TYPE U_NCI_R_PARAMETER_I :
UNION

  stCtrl              : ARRAY[1..MAX_NCI_CH] OF ST_R_Parameter;

  byCtrl    AT %q*    : ARRAY[1..MAX_NCI_CH] OF
                        ARRAY[1..SIZEOF(ST_R_Parameter)] OF BYTE;
END_UNION
END_TYPE

(* stored: Version 1.1.0.1
   DUT U_NCI_R_PARAMETER_I: Id {195e8a25-bcd7-43b7-b5c5-7df26282d8f3} *)
